// TIA Portal V20 export
TYPE "type_emRelations_em5_sequence"
// stored: Access Published, Namespace Unit1
   STRUCT
      transferPnPLeft : Struct
         jobs : "LAF_typeJobs";
         sequence : "LAF_typeSequence";
         selectJobStatus { S7_SetPoint := 'True'} : Array[0..10] of "LAF_typeJobStatus";
         "step" : "LER_typeStep";
         jobInterface : Struct
            sideTapePICKJob2_A : "LER_typeJobInterface";
            hotPressLeftPLACEJob3_A : "LER_typeJobInterface";
            hotPressLeftPICKJob4_A : "LER_typeJobInterface";
            sideTapePICKJob5_B : "LER_typeJobInterface";
            hotPressRightPLACEJob6_B : "LER_typeJobInterface";
            hotPressRightPICKJob7_B : "LER_typeJobInterface";
            hipotThicknessPLACEJob9 : "LER_typeJobInterface";
         END_STRUCT;
         homeCheck : Struct
            waitPosPartNoDetect { ExternalWritable := 'False'} : Bool;
            waitPosPartDetect { ExternalWritable := 'False'} : Bool;
            sideTapePosPartNoDetect { ExternalWritable := 'False'} : Bool;
            sideTapePosPartDetect { ExternalWritable := 'False'} : Bool;
            hotPressLeftPosPartNoDetect { ExternalWritable := 'False'} : Bool;
            hotPressLeftPosPartDetect { ExternalWritable := 'False'} : Bool;
            hotPressRightPosPartNoDetect { ExternalWritable := 'False'} : Bool;
            hotPressRightPosPartDetect { ExternalWritable := 'False'} : Bool;
            hipotThicknessPosPartNoDetect { ExternalWritable := 'False'} : Bool;
            hipotThicknessPosPartDetect { ExternalWritable := 'False'} : Bool;
            defaultPosPartDetect : Bool;
            defaultPosPartNoDetect : Bool;
         END_STRUCT;
      END_STRUCT;
      transferPnPRight : Struct
         jobs : "LAF_typeJobs";
         sequence : "LAF_typeSequence";
         selectJobStatus { S7_SetPoint := 'True'} : Array[0..10] of "LAF_typeJobStatus";
         "step" : "LER_typeStep";
         jobInterface : Struct
            hipotThicknessPICKJob2 : "LER_typeJobInterface";
            visionPLACEJob3 : "LER_typeJobInterface";
            visionPICKJob4 : "LER_typeJobInterface";
            laserMarkPLACEJob5 : "LER_typeJobInterface";
            laserMarkPICKJob6 : "LER_typeJobInterface";
            weightCheckPLACEJob9 : "LER_typeJobInterface";
         END_STRUCT;
         homeCheck : Struct
            waitPosPartNoDetect { ExternalWritable := 'False'} : Bool;
            waitPosPartDetect { ExternalWritable := 'False'} : Bool;
            hipotThicknessPosPartNoDetect { ExternalWritable := 'False'} : Bool;
            hipotThicknessPosPartDetect { ExternalWritable := 'False'} : Bool;
            visionPosPartNoDetect { ExternalWritable := 'False'} : Bool;
            visionPosPartDetect { ExternalWritable := 'False'} : Bool;
            laserMarkPosPartNoDetect { ExternalWritable := 'False'} : Bool;
            laserMarkPosPartDetect { ExternalWritable := 'False'} : Bool;
            weightCheckPosPartNoDetect { ExternalWritable := 'False'} : Bool;
            weightCheckPosPartDetect { ExternalWritable := 'False'} : Bool;
            defaultPosPartDetect : Bool;
            defaultPosPartNoDetect : Bool;
         END_STRUCT;
      END_STRUCT;
      GRnR_TransferPnP : Struct
         jobs : "LAF_typeJobs";
         sequence : "LAF_typeSequence";
         selectJobStatus { S7_SetPoint := 'True'} : Array[0..10] of "LAF_typeJobStatus";
         "step" : "LER_typeStep";
         jobInterface : Struct
            transferPnPLeft : Struct
               sideTapePICKJob2 : "LER_typeJobInterface";
               hipotThicknessPLACEJob3 : "LER_typeJobInterface";
               hipotThicknessPICKJob4 : "LER_typeJobInterface";
            END_STRUCT;
            transferPnPRight : Struct
               hipotThicknessPICKJob5 : "LER_typeJobInterface";
               visionPLACEJob6 : "LER_typeJobInterface";
               visionPICKJob7 : "LER_typeJobInterface";
               weightCheckPLACEJob8 : "LER_typeJobInterface";
               weightCheckPICKJob9 : "LER_typeJobInterface";
            END_STRUCT;
         END_STRUCT;
      END_STRUCT;
   END_STRUCT;
   // // transferPnPLeft."step".action1[101] : Step[101] : JOB[1] Condition
   // // transferPnPLeft."step".action1[110] : Step[110] : Transfer PP Left Clamp Open
   // // transferPnPLeft."step".action1[130] : Step[130] : Transfer PP Left Clamp Close
   // // transferPnPLeft."step".action1[160] : Step[160] : Transfer PP Left Y-Axis Wait Pos
   // // transferPnPLeft."step".action1[170] : Step[170] : Transfer PP Left Z-Axis Wait Pos
   // // transferPnPLeft."step".action1[180] : Step[180] : Transfer PP Left X-Axis Wait Pos
   // // transferPnPLeft."step".action1[190] : Step[190] : JOB[1] Step End
   // // transferPnPLeft."step".action1[201] : Step[201] : JOB[2] Condition
   // // transferPnPLeft."step".action1[210] : Step[210] : Transfer PP Left X/Z-Axis Side Tape Pos
   // // transferPnPLeft."step".action1[230] : Step[230] : Transfer PP Left Y-Axis Side Tape Pos
   // // transferPnPLeft."step".action1[240] : Step[240] : Transfer PP Left Clamp Close
   // // transferPnPLeft."step".action1[242] : Step[242] : Transfer PP Left [Unclamp request] => Side Tape Fix Stage
   // // transferPnPLeft."step".action1[280] : Step[280] : Transfer PP Left Y-Axis Wait Pos
   // // transferPnPLeft."step".action1[290] : Step[290] : JOB[2] Step End
   // // transferPnPLeft."step".action1[301] : Step[301] : JOB[3] Condition
   // // transferPnPLeft."step".action1[310] : Step[310] : Transfer PP Left X/Z-Axis Hot Press Left Pos
   // // transferPnPLeft."step".action1[330] : Step[330] : Transfer PP Left Y-Axis Hot Press Left Pos
   // // transferPnPLeft."step".action1[340] : Step[340] : Transfer PP Left [Lift Up Request] => Hot Press Left
   // // transferPnPLeft."step".action1[350] : Step[350] : Transfer PP Left Clamp Open
   // // transferPnPLeft."step".action1[380] : Step[380] : Transfer PP Left Y-Axis Wait Pos
   // // transferPnPLeft."step".action1[390] : Step[390] : JOB[3] Step End
   // // transferPnPLeft."step".action1[401] : Step[401] : JOB[4] Condition
   // // transferPnPLeft."step".action1[410] : Step[410] : Transfer PP Left X/Z-Axis Hot Press Left Pos
   // // transferPnPLeft."step".action1[430] : Step[430] : Transfer PP Left Y-Axis Hot Press Left Pos
   // // transferPnPLeft."step".action1[440] : Step[440] : Transfer PP Left Clamp Close
   // // transferPnPLeft."step".action1[480] : Step[480] : Transfer PP Left Y-Axis Wait Pos
   // // transferPnPLeft."step".action1[490] : Step[490] : JOB[4] Step End
   // // transferPnPLeft."step".action1[501] : Step[501] : JOB[5] Condition
   // // transferPnPLeft."step".action1[510] : Step[510] : Transfer PP Left X/Z-Axis Side Tape Pos
   // // transferPnPLeft."step".action1[530] : Step[530] : Transfer PP Left Y-Axis Side Tape Pos
   // // transferPnPLeft."step".action1[540] : Step[540] : Transfer PP Left Clamp Close
   // // transferPnPLeft."step".action1[542] : Step[542] : Transfer PP Left [Unclamp request] => Side Tape Fix Stage
   // // transferPnPLeft."step".action1[580] : Step[580] : Transfer PP Left Y-Axis Wait Pos
   // // transferPnPLeft."step".action1[590] : Step[590] : JOB[5] Step End
   // // transferPnPLeft."step".action1[601] : Step[601] : JOB[6] Condition
   // // transferPnPLeft."step".action1[610] : Step[610] : Transfer PP Left X/Z-Axis Hot Press Right Pos
   // // transferPnPLeft."step".action1[630] : Step[630] : Transfer PP Left Y-Axis Hot Press Right Pos
   // // transferPnPLeft."step".action1[640] : Step[640] : Transfer PP Left [Lift Up Request] => Hot Press Right
   // // transferPnPLeft."step".action1[650] : Step[650] : Transfer PP Left Clamp Open
   // // transferPnPLeft."step".action1[680] : Step[680] : Transfer PP Left Y-Axis Wait Pos
   // // transferPnPLeft."step".action1[690] : Step[690] : JOB[6] Step End
   // // transferPnPLeft."step".action1[701] : Step[701] : JOB[7] Condition
   // // transferPnPLeft."step".action1[710] : Step[710] : Transfer PP Left X/Z-Axis Hot Press Right Pos
   // // transferPnPLeft."step".action1[730] : Step[730] : Transfer PP Left Y-Axis Hot Press Right Pos
   // // transferPnPLeft."step".action1[740] : Step[740] : Transfer PP Left Clamp Close
   // // transferPnPLeft."step".action1[780] : Step[780] : Transfer PP Left Y-Axis Wait Pos
   // // transferPnPLeft."step".action1[790] : Step[790] : JOB[7] Step End
   // // transferPnPLeft."step".action1[901] : Step[901] : JOB[9] Condition
   // // transferPnPLeft."step".action1[910] : Step[910] : Transfer PP Left X/Z-Axis Hipot & Thickness Pos
   // // transferPnPLeft."step".action1[930] : Step[930] : Transfer PP Left Y-Axis Hipot & Thickness Pos
   // // transferPnPLeft."step".action1[940] : Step[940] : Transfer PP Left [Lift Up Request] => Hipot & Thickness
   // // transferPnPLeft."step".action1[950] : Step[950] : Transfer PP Left Clamp Open
   // // transferPnPLeft."step".action1[980] : Step[980] : Transfer PP Left Y-Axis Wait Pos
   // // transferPnPLeft."step".action1[981] : Step[981] : Transfer PP Left X/Z-Axis Wait Pos
   // // transferPnPLeft."step".action1[990] : Step[990] : JOB[9] Step End
   // // transferPnPLeft."step".transition1[101] : Step[101] : JOB[1] Condition
   // // transferPnPLeft."step".transition1[110] : Step[110] : Transfer PP Left Clamp Open
   // // transferPnPLeft."step".transition1[130] : Step[130] : Transfer PP Left Clamp Close
   // // transferPnPLeft."step".transition1[160] : Step[160] : Transfer PP Left Y-Axis Wait Pos
   // // transferPnPLeft."step".transition1[170] : Step[170] : Transfer PP Left Z-Axis Wait Pos
   // // transferPnPLeft."step".transition1[180] : Step[180] : Transfer PP Left X-Axis Wait Pos
   // // transferPnPLeft."step".transition1[190] : Step[190] : JOB[1] Step End
   // // transferPnPLeft."step".transition1[201] : Step[201] : JOB[2] Condition
   // // transferPnPLeft."step".transition1[210] : Step[210] : Transfer PP Left X/Z-Axis Side Tape Pos
   // // transferPnPLeft."step".transition1[230] : Step[230] : Transfer PP Left Y-Axis Side Tape Pos
   // // transferPnPLeft."step".transition1[240] : Step[240] : Transfer PP Left Clamp Close
   // // transferPnPLeft."step".transition1[242] : Step[242] : Transfer PP Left [Unclamp request] => Side Tape Fix Stage
   // // transferPnPLeft."step".transition1[280] : Step[280] : Transfer PP Left Y-Axis Wait Pos
   // // transferPnPLeft."step".transition1[290] : Step[290] : JOB[2] Step End
   // // transferPnPLeft."step".transition1[301] : Step[301] : JOB[3] Condition
   // // transferPnPLeft."step".transition1[310] : Step[310] : Transfer PP Left X/Z-Axis Hot Press Left Pos
   // // transferPnPLeft."step".transition1[330] : Step[330] : Transfer PP Left Y-Axis Hot Press Left Pos
   // // transferPnPLeft."step".transition1[340] : Step[340] : Transfer PP Left [Lift Up Request] => Hot Press Left
   // // transferPnPLeft."step".transition1[350] : Step[350] : Transfer PP Left Clamp Open
   // // transferPnPLeft."step".transition1[380] : Step[380] : Transfer PP Left Y-Axis Wait Pos
   // // transferPnPLeft."step".transition1[390] : Step[390] : JOB[3] Step End
   // // transferPnPLeft."step".transition1[401] : Step[401] : JOB[4] Condition
   // // transferPnPLeft."step".transition1[410] : Step[410] : Transfer PP Left X/Z-Axis Hot Press Left Pos
   // // transferPnPLeft."step".transition1[430] : Step[430] : Transfer PP Left Y-Axis Hot Press Left Pos
   // // transferPnPLeft."step".transition1[440] : Step[440] : Transfer PP Left Clamp Close
   // // transferPnPLeft."step".transition1[480] : Step[480] : Transfer PP Left Y-Axis Wait Pos
   // // transferPnPLeft."step".transition1[490] : Step[490] : JOB[4] Step End
   // // transferPnPLeft."step".transition1[501] : Step[501] : JOB[5] Condition
   // // transferPnPLeft."step".transition1[510] : Step[510] : Transfer PP Left X/Z-Axis Side Tape Pos
   // // transferPnPLeft."step".transition1[530] : Step[530] : Transfer PP Left Y-Axis Side Tape Pos
   // // transferPnPLeft."step".transition1[540] : Step[540] : Transfer PP Left Clamp Close
   // // transferPnPLeft."step".transition1[542] : Step[542] : Transfer PP Left [Unclamp request] => Side Tape Fix Stage
   // // transferPnPLeft."step".transition1[580] : Step[580] : Transfer PP Left Y-Axis Wait Pos
   // // transferPnPLeft."step".transition1[590] : Step[590] : JOB[5] Step End
   // // transferPnPLeft."step".transition1[601] : Step[601] : JOB[6] Condition
   // // transferPnPLeft."step".transition1[610] : Step[610] : Transfer PP Left X/Z-Axis Hot Press Right Pos
   // // transferPnPLeft."step".transition1[630] : Step[630] : Transfer PP Left Y-Axis Hot Press Right Pos
   // // transferPnPLeft."step".transition1[640] : Step[640] : Transfer PP Left [Lift Up Request] => Hot Press Right
   // // transferPnPLeft."step".transition1[650] : Step[650] : Transfer PP Left Clamp Open
   // // transferPnPLeft."step".transition1[680] : Step[680] : Transfer PP Left Y-Axis Wait Pos
   // // transferPnPLeft."step".transition1[690] : Step[690] : JOB[6] Step End
   // // transferPnPLeft."step".transition1[701] : Step[701] : JOB[7] Condition
   // // transferPnPLeft."step".transition1[710] : Step[710] : Transfer PP Left X/Z-Axis Hot Press Right Pos
   // // transferPnPLeft."step".transition1[730] : Step[730] : Transfer PP Left Y-Axis Hot Press Right Pos
   // // transferPnPLeft."step".transition1[740] : Step[740] : Transfer PP Left Clamp Close
   // // transferPnPLeft."step".transition1[780] : Step[780] : Transfer PP Left Y-Axis Wait Pos
   // // transferPnPLeft."step".transition1[790] : Step[790] : JOB[7] Step End
   // // transferPnPLeft."step".transition1[901] : Step[901] : JOB[9] Condition
   // // transferPnPLeft."step".transition1[910] : Step[910] : Transfer PP Left X/Z-Axis Hipot & Thickness Pos
   // // transferPnPLeft."step".transition1[930] : Step[930] : Transfer PP Left Y-Axis Hipot & Thickness Pos
   // // transferPnPLeft."step".transition1[940] : Step[940] : Transfer PP Left [Lift Up Request] => Hipot & Thickness
   // // transferPnPLeft."step".transition1[950] : Step[950] : Transfer PP Left Clamp Open
   // // transferPnPLeft."step".transition1[980] : Step[980] : Transfer PP Left Y-Axis Wait Pos
   // // transferPnPLeft."step".transition1[981] : Step[981] : Transfer PP Left X/Z-Axis Wait Pos
   // // transferPnPLeft."step".transition1[990] : Step[990] : JOB[9] Step End
   // // transferPnPRight."step".action1[101] : Step[101] : JOB[1] Condition
   // // transferPnPRight."step".action1[110] : Step[110] : Transfer PP Right Clamp Open
   // // transferPnPRight."step".action1[130] : Step[130] : Transfer PP Right Clamp Close
   // // transferPnPRight."step".action1[160] : Step[160] : Transfer PP Right Y-Axis Wait Position
   // // transferPnPRight."step".action1[170] : Step[170] : Transfer PP Right Z-Axis Wait Position
   // // transferPnPRight."step".action1[180] : Step[180] : Transfer PP Right X-Axis Wait Position
   // // transferPnPRight."step".action1[190] : Step[190] : JOB[1] Step End
   // // transferPnPRight."step".action1[201] : Step[201] : JOB[2] Condition
   // // transferPnPRight."step".action1[210] : Step[210] : Transfer PP Right X/Z-Axis Hipot & Thickness Pos
   // // transferPnPRight."step".action1[230] : Step[230] : Transfer PP Right Y-Axis Hipot & Thickness Pos
   // // transferPnPRight."step".action1[240] : Step[240] : Transfer PP Right Clamp Close
   // // transferPnPRight."step".action1[280] : Step[280] : Transfer PP Right Y-Axis Wait Pos
   // // transferPnPRight."step".action1[290] : Step[290] : JOB[2] Step End
   // // transferPnPRight."step".action1[301] : Step[301] : JOB[3] Condition
   // // transferPnPRight."step".action1[310] : Step[310] : Transfer PP Right X/Z-Axis Vision Pos
   // // transferPnPRight."step".action1[330] : Step[330] : Transfer PP Right Y-Axis Vision Pos
   // // transferPnPRight."step".action1[340] : Step[340] : Transfer PP Right [Lift Up Request] => Vision Check
   // // transferPnPRight."step".action1[350] : Step[350] : Transfer PP Right Clamp Open
   // // transferPnPRight."step".action1[380] : Step[380] : Transfer PP Right Y-Axis Wait Pos
   // // transferPnPRight."step".action1[390] : Step[390] : JOB[3] Step End
   // // transferPnPRight."step".action1[401] : Step[401] : JOB[4] Condition
   // // transferPnPRight."step".action1[410] : Step[410] : Transfer PP Right X/Z-Axis Vision Pos
   // // transferPnPRight."step".action1[430] : Step[430] : Transfer PP Right Y-Axis Vision Pos
   // // transferPnPRight."step".action1[440] : Step[440] : Transfer PP Right Clamp Close
   // // transferPnPRight."step".action1[480] : Step[480] : Transfer PP Right Y-Axis Wait Pos
   // // transferPnPRight."step".action1[490] : Step[490] : JOB[4] Step End
   // // transferPnPRight."step".action1[501] : Step[501] : JOB[5] Condition
   // // transferPnPRight."step".action1[510] : Step[510] : Transfer PP Right X/Z-Axis Laser Mark Pos
   // // transferPnPRight."step".action1[530] : Step[530] : Transfer PP Right Y-Axis Laser Mark Pos
   // // transferPnPRight."step".action1[540] : Step[540] : Transfer PP Right [Lift Up Request] => Laser Mark
   // // transferPnPRight."step".action1[550] : Step[550] : Transfer PP Right Clamp Open
   // // transferPnPRight."step".action1[580] : Step[580] : Transfer PP Right Y-Axis Wait Pos
   // // transferPnPRight."step".action1[590] : Step[590] : JOB[5] Step End
   // // transferPnPRight."step".action1[601] : Step[601] : JOB[6] Condition
   // // transferPnPRight."step".action1[602] : Step[602] : QR Read Start
   // // transferPnPRight."step".action1[603] : Step[603] : QR Read Result
   // // transferPnPRight."step".action1[604] : Step[604] : QR Read Start [NG]
   // // transferPnPRight."step".action1[605] : Step[605] : QR Read Result [NG]
   // // transferPnPRight."step".action1[610] : Step[610] : Transfer PP Right X/Z-Axis Laser Mark Pos
   // // transferPnPRight."step".action1[630] : Step[630] : Transfer PP Right Y-Axis Laser Mark Pos
   // // transferPnPRight."step".action1[640] : Step[640] : Transfer PP Right Clamp Close
   // // transferPnPRight."step".action1[680] : Step[680] : Transfer PP Right Y-Axis Wait Pos
   // // transferPnPRight."step".action1[690] : Step[690] : JOB[6] Step End
   // // transferPnPRight."step".action1[701] : Step[701] : JOB[7] Condition
   // // transferPnPRight."step".action1[710] : Step[710] : Transfer PP Right X/Z-Axis Laser Mark Pos
   // // transferPnPRight."step".action1[730] : Step[730] : Transfer PP Right Y-Axis Laser Mark Pos
   // // transferPnPRight."step".action1[740] : Step[740] : Transfer PP Right [Lift Up Request] => Laser Mark
   // // transferPnPRight."step".action1[750] : Step[750] : Transfer PP Right Clamp Open
   // // transferPnPRight."step".action1[780] : Step[780] : Transfer PP Right Y-Axis Wait Pos
   // // transferPnPRight."step".action1[790] : Step[790] : JOB[7] Step End
   // // transferPnPRight."step".action1[801] : Step[801] : JOB[8] Condition
   // // transferPnPRight."step".action1[810] : Step[810] : Transfer PP Right X/Z-Axis Laser Mark Pos
   // // transferPnPRight."step".action1[830] : Step[830] : Transfer PP Right Y-Axis Laser Mark Pos
   // // transferPnPRight."step".action1[840] : Step[840] : Transfer PP Right Clamp Close
   // // transferPnPRight."step".action1[880] : Step[880] : Transfer PP Right Y-Axis Wait Pos
   // // transferPnPRight."step".action1[890] : Step[890] : JOB[8] Step End
   // // transferPnPRight."step".action1[901] : Step[901] : JOB[9] Condition
   // // transferPnPRight."step".action1[910] : Step[910] : Transfer PP Right X/Z-Axis Weight Check Pos
   // // transferPnPRight."step".action1[930] : Step[930] : Transfer PP Right Y-Axis Weight Check Pos
   // // transferPnPRight."step".action1[931] : Step[931] : Transfer PP Right Z-Axis Weight Check Pos
   // // transferPnPRight."step".action1[940] : Step[940] : Transfer PP Right [Lift Up Request] => Weight Check
   // // transferPnPRight."step".action1[950] : Step[950] : Transfer PP Right Clamp Open
   // // transferPnPRight."step".action1[980] : Step[980] : Transfer PP Right Y-Axis Wait Pos
   // // transferPnPRight."step".action1[981] : Step[981] : Transfer PP Right X/Z-Axis Wait Pos
   // // transferPnPRight."step".action1[990] : Step[990] : JOB[9] Step End
   // // transferPnPRight."step".transition1[101] : Step[101] : JOB[1] Condition
   // // transferPnPRight."step".transition1[110] : Step[110] : Transfer PP Right Clamp Open
   // // transferPnPRight."step".transition1[130] : Step[130] : Transfer PP Right Clamp Close
   // // transferPnPRight."step".transition1[160] : Step[160] : Transfer PP Right Y-Axis Wait Position
   // // transferPnPRight."step".transition1[170] : Step[170] : Transfer PP Right Z-Axis Wait Position
   // // transferPnPRight."step".transition1[180] : Step[180] : Transfer PP Right X-Axis Wait Position
   // // transferPnPRight."step".transition1[190] : Step[190] : JOB[1] Step End
   // // transferPnPRight."step".transition1[201] : Step[201] : JOB[2] Condition
   // // transferPnPRight."step".transition1[210] : Step[210] : Transfer PP Right X/Z-Axis Hipot & Thickness Pos
   // // transferPnPRight."step".transition1[230] : Step[230] : Transfer PP Right Y-Axis Hipot & Thickness Pos
   // // transferPnPRight."step".transition1[240] : Step[240] : Transfer PP Right Clamp Close
   // // transferPnPRight."step".transition1[280] : Step[280] : Transfer PP Right Y-Axis Wait Pos
   // // transferPnPRight."step".transition1[290] : Step[290] : JOB[2] Step End
   // // transferPnPRight."step".transition1[301] : Step[301] : JOB[3] Condition
   // // transferPnPRight."step".transition1[310] : Step[310] : Transfer PP Right X/Z-Axis Vision Pos
   // // transferPnPRight."step".transition1[330] : Step[330] : Transfer PP Right Y-Axis Vision Pos
   // // transferPnPRight."step".transition1[340] : Step[340] : Transfer PP Right [Lift Up Request] => Vision Check
   // // transferPnPRight."step".transition1[350] : Step[350] : Transfer PP Right Clamp Open
   // // transferPnPRight."step".transition1[380] : Step[380] : Transfer PP Right Y-Axis Wait Pos
   // // transferPnPRight."step".transition1[390] : Step[390] : JOB[3] Step End
   // // transferPnPRight."step".transition1[401] : Step[401] : JOB[4] Condition
   // // transferPnPRight."step".transition1[410] : Step[410] : Transfer PP Right X/Z-Axis Vision Pos
   // // transferPnPRight."step".transition1[430] : Step[430] : Transfer PP Right Y-Axis Vision Pos
   // // transferPnPRight."step".transition1[440] : Step[440] : Transfer PP Right Clamp Close
   // // transferPnPRight."step".transition1[480] : Step[480] : Transfer PP Right Y-Axis Wait Pos
   // // transferPnPRight."step".transition1[490] : Step[490] : JOB[4] Step End
   // // transferPnPRight."step".transition1[501] : Step[501] : JOB[5] Condition
   // // transferPnPRight."step".transition1[510] : Step[510] : Transfer PP Right X/Z-Axis Laser Mark Pos
   // // transferPnPRight."step".transition1[530] : Step[530] : Transfer PP Right Y-Axis Laser Mark Pos
   // // transferPnPRight."step".transition1[540] : Step[540] : Transfer PP Right [Lift Up Request] => Laser Mark
   // // transferPnPRight."step".transition1[550] : Step[550] : Transfer PP Right Clamp Open
   // // transferPnPRight."step".transition1[580] : Step[580] : Transfer PP Right Y-Axis Wait Pos
   // // transferPnPRight."step".transition1[590] : Step[590] : JOB[5] Step End
   // // transferPnPRight."step".transition1[601] : Step[601] : JOB[6] Condition
   // // transferPnPRight."step".transition1[602] : Step[602] : QR Read Start
   // // transferPnPRight."step".transition1[603] : Step[603] : QR Read Result
   // // transferPnPRight."step".transition1[604] : Step[604] : QR Read Start [NG]
   // // transferPnPRight."step".transition1[605] : Step[605] : QR Read Result [NG]
   // // transferPnPRight."step".transition1[610] : Step[610] : Transfer PP Right X/Z-Axis Laser Mark Pos
   // // transferPnPRight."step".transition1[630] : Step[630] : Transfer PP Right Y-Axis Laser Mark Pos
   // // transferPnPRight."step".transition1[640] : Step[640] : Transfer PP Right Clamp Close
   // // transferPnPRight."step".transition1[680] : Step[680] : Transfer PP Right Y-Axis Wait Pos
   // // transferPnPRight."step".transition1[690] : Step[690] : JOB[6] Step End
   // // transferPnPRight."step".transition1[701] : Step[701] : JOB[7] Condition
   // // transferPnPRight."step".transition1[710] : Step[710] : Transfer PP Right X/Z-Axis Laser Mark Pos
   // // transferPnPRight."step".transition1[730] : Step[730] : Transfer PP Right Y-Axis Laser Mark Pos
   // // transferPnPRight."step".transition1[740] : Step[740] : Transfer PP Right [Lift Up Request] => Laser Mark
   // // transferPnPRight."step".transition1[750] : Step[750] : Transfer PP Right Clamp Open
   // // transferPnPRight."step".transition1[780] : Step[780] : Transfer PP Right Y-Axis Wait Pos
   // // transferPnPRight."step".transition1[790] : Step[790] : JOB[7] Step End
   // // transferPnPRight."step".transition1[801] : Step[801] : JOB[8] Condition
   // // transferPnPRight."step".transition1[810] : Step[810] : Transfer PP Right X/Z-Axis Laser Mark Pos
   // // transferPnPRight."step".transition1[830] : Step[830] : Transfer PP Right Y-Axis Laser Mark Pos
   // // transferPnPRight."step".transition1[840] : Step[840] : Transfer PP Right Clamp Close
   // // transferPnPRight."step".transition1[880] : Step[880] : Transfer PP Right Y-Axis Wait Pos
   // // transferPnPRight."step".transition1[890] : Step[890] : JOB[8] Step End
   // // transferPnPRight."step".transition1[901] : Step[901] : JOB[9] Condition
   // // transferPnPRight."step".transition1[910] : Step[910] : Transfer PP Right X/Z-Axis Weight Check Pos
   // // transferPnPRight."step".transition1[930] : Step[930] : Transfer PP Right Y-Axis Weight Check Pos
   // // transferPnPRight."step".transition1[931] : Step[931] : Transfer PP Right Z-Axis Weight Check Pos
   // // transferPnPRight."step".transition1[940] : Step[940] : Transfer PP Right [Lift Up Request] => Weight Check
   // // transferPnPRight."step".transition1[950] : Step[950] : Transfer PP Right Clamp Open
   // // transferPnPRight."step".transition1[980] : Step[980] : Transfer PP Right Y-Axis Wait Pos
   // // transferPnPRight."step".transition1[981] : Step[981] : Transfer PP Right X/Z-Axis Wait Pos
   // // transferPnPRight."step".transition1[990] : Step[990] : JOB[9] Step End
   // // GRnR_TransferPnP."step".action1[201] : Step[201] : JOB[2] Condition
   // // GRnR_TransferPnP."step".action1[210] : Step[210] : Transfer PP Left X/Z-Axis Side Tape Pos
   // // GRnR_TransferPnP."step".action1[230] : Step[230] : Transfer PP Left Y-Axis Side Tape Pos
   // // GRnR_TransferPnP."step".action1[240] : Step[240] : Transfer PP Left Clamp Close
   // // GRnR_TransferPnP."step".action1[241] : Step[241] : Transfer PP Left [Unclamp request] => Side Tape Fix Stage
   // // GRnR_TransferPnP."step".action1[280] : Step[280] : Transfer PP Left Y-Axis Wait Pos
   // // GRnR_TransferPnP."step".action1[290] : Step[290] : JOB[2] Step End
   // // GRnR_TransferPnP."step".action1[301] : Step[301] : JOB[3] Condition
   // // GRnR_TransferPnP."step".action1[310] : Step[310] : Transfer PP Left X/Z-Axis Hipot & Thickness Pos
   // // GRnR_TransferPnP."step".action1[330] : Step[330] : Transfer PP Left Y-Axis Hipot & Thickness Pos
   // // GRnR_TransferPnP."step".action1[340] : Step[340] : Transfer PP Left [Lift Up Request] => Hipot & Thickness
   // // GRnR_TransferPnP."step".action1[350] : Step[350] : Transfer PP Left Clamp Open
   // // GRnR_TransferPnP."step".action1[380] : Step[380] : Transfer PP Left Y-Axis Wait Pos
   // // GRnR_TransferPnP."step".action1[381] : Step[381] : Transfer PP Left X/Z-Axis Wait Pos
   // // GRnR_TransferPnP."step".action1[390] : Step[390] : JOB[3] Step End
   // // GRnR_TransferPnP."step".action1[401] : Step[401] : JOB[4] Condition
   // // GRnR_TransferPnP."step".action1[410] : Step[410] : Transfer PP Left X/Z-Axis Hipot & Thickness Pos
   // // GRnR_TransferPnP."step".action1[430] : Step[430] : Transfer PP Left Y-Axis Hipot & Thickness Pos
   // // GRnR_TransferPnP."step".action1[440] : Step[440] : Transfer PP Left Clamp Close
   // // GRnR_TransferPnP."step".action1[480] : Step[480] : Transfer PP Left Y-Axis Wait Pos
   // // GRnR_TransferPnP."step".action1[481] : Step[481] : Transfer PP Left X/Z-Axis Wait Pos
   // // GRnR_TransferPnP."step".action1[490] : Step[490] : JOB[4] Step End
   // // GRnR_TransferPnP."step".action1[501] : Step[501] : JOB[5] Condition
   // // GRnR_TransferPnP."step".action1[510] : Step[510] : Transfer PP Right X/Z-Axis Hipot & Thickness Pos
   // // GRnR_TransferPnP."step".action1[530] : Step[530] : Transfer PP Right Y-Axis Hipot & Thickness Pos
   // // GRnR_TransferPnP."step".action1[540] : Step[540] : Transfer PP Right Clamp Close
   // // GRnR_TransferPnP."step".action1[580] : Step[580] : Transfer PP Right Y-Axis Wait Pos
   // // GRnR_TransferPnP."step".action1[590] : Step[590] : JOB[5] Step End
   // // GRnR_TransferPnP."step".action1[601] : Step[601] : JOB[6] Condition
   // // GRnR_TransferPnP."step".action1[610] : Step[610] : Transfer PP Right X/Z-Axis Vision Pos
   // // GRnR_TransferPnP."step".action1[630] : Step[630] : Transfer PP Right Y-Axis Vision Pos
   // // GRnR_TransferPnP."step".action1[640] : Step[640] : Transfer PP Right [Lift Up Request] => Vision Check
   // // GRnR_TransferPnP."step".action1[650] : Step[650] : Transfer PP Right Clamp Open
   // // GRnR_TransferPnP."step".action1[680] : Step[680] : Transfer PP Right Y-Axis Wait Pos
   // // GRnR_TransferPnP."step".action1[690] : Step[690] : JOB[6] Step End
   // // GRnR_TransferPnP."step".action1[701] : Step[701] : JOB[7] Condition
   // // GRnR_TransferPnP."step".action1[710] : Step[710] : Transfer PP Right X/Z-Axis Vision Pos
   // // GRnR_TransferPnP."step".action1[730] : Step[730] : Transfer PP Right Y-Axis Vision Pos
   // // GRnR_TransferPnP."step".action1[740] : Step[740] : Transfer PP Right Clamp Close
   // // GRnR_TransferPnP."step".action1[780] : Step[780] : Transfer PP Right Y-Axis Wait Pos
   // // GRnR_TransferPnP."step".action1[790] : Step[790] : JOB[7] Step End
   // // GRnR_TransferPnP."step".action1[801] : Step[801] : JOB[8] Condition
   // // GRnR_TransferPnP."step".action1[810] : Step[810] : Transfer PP Right X/Z-Axis Weight Check Pos
   // // GRnR_TransferPnP."step".action1[830] : Step[830] : Transfer PP Right Y-Axis Weight Check Pos
   // // GRnR_TransferPnP."step".action1[831] : Step[831] : Transfer PP Right Z-Axis Weight Check Pos
   // // GRnR_TransferPnP."step".action1[840] : Step[840] : Transfer PP Right [Lift Up Request] => Weight Check
   // // GRnR_TransferPnP."step".action1[850] : Step[850] : Transfer PP Right Clamp Open
   // // GRnR_TransferPnP."step".action1[880] : Step[880] : Transfer PP Right Y-Axis Wait Pos
   // // GRnR_TransferPnP."step".action1[881] : Step[881] : Transfer PP Right X/Z-Axis Wait Pos
   // // GRnR_TransferPnP."step".action1[890] : Step[890] : JOB[8] Step End
   // // GRnR_TransferPnP."step".action1[901] : Step[901] : JOB[9] Condition
   // // GRnR_TransferPnP."step".action1[910] : Step[910] : Transfer PP Right X/Z-Axis Weight Check Pos
   // // GRnR_TransferPnP."step".action1[930] : Step[930] : Transfer PP Right Y-Axis Weight Pos
   // // GRnR_TransferPnP."step".action1[940] : Step[940] : Transfer PP Right Clamp Close
   // // GRnR_TransferPnP."step".transition1[201] : Step[201] : JOB[2] Condition
   // // GRnR_TransferPnP."step".transition1[210] : Step[210] : Transfer PP Left X/Z-Axis Side Tape Pos
   // // GRnR_TransferPnP."step".transition1[230] : Step[230] : Transfer PP Left Y-Axis Side Tape Pos
   // // GRnR_TransferPnP."step".transition1[240] : Step[240] : Transfer PP Left Clamp Close
   // // GRnR_TransferPnP."step".transition1[241] : Step[241] : Transfer PP Left [Unclamp request] => Side Tape Fix Stage
   // // GRnR_TransferPnP."step".transition1[280] : Step[280] : Transfer PP Left Y-Axis Wait Pos
   // // GRnR_TransferPnP."step".transition1[290] : Step[290] : JOB[2] Step End
   // // GRnR_TransferPnP."step".transition1[301] : Step[301] : JOB[3] Condition
   // // GRnR_TransferPnP."step".transition1[310] : Step[310] : Transfer PP Left X/Z-Axis Hipot & Thickness Pos
   // // GRnR_TransferPnP."step".transition1[330] : Step[330] : Transfer PP Left Y-Axis Hipot & Thickness Pos
   // // GRnR_TransferPnP."step".transition1[340] : Step[340] : Transfer PP Left [Lift Up Request] => Hipot & Thickness
   // // GRnR_TransferPnP."step".transition1[350] : Step[350] : Transfer PP Left Clamp Open
   // // GRnR_TransferPnP."step".transition1[380] : Step[380] : Transfer PP Left Y-Axis Wait Pos
   // // GRnR_TransferPnP."step".transition1[381] : Step[381] : Transfer PP Left X/Z-Axis Wait Pos
   // // GRnR_TransferPnP."step".transition1[390] : Step[390] : JOB[3] Step End
   // // GRnR_TransferPnP."step".transition1[401] : Step[401] : JOB[4] Condition
   // // GRnR_TransferPnP."step".transition1[410] : Step[410] : Transfer PP Left X/Z-Axis Hipot & Thickness Pos
   // // GRnR_TransferPnP."step".transition1[430] : Step[430] : Transfer PP Left Y-Axis Hipot & Thickness Pos
   // // GRnR_TransferPnP."step".transition1[440] : Step[440] : Transfer PP Left Clamp Close
   // // GRnR_TransferPnP."step".transition1[480] : Step[480] : Transfer PP Left Y-Axis Wait Pos
   // // GRnR_TransferPnP."step".transition1[481] : Step[481] : Transfer PP Left X/Z-Axis Wait Pos
   // // GRnR_TransferPnP."step".transition1[490] : Step[490] : JOB[4] Step End
   // // GRnR_TransferPnP."step".transition1[501] : Step[501] : JOB[5] Condition
   // // GRnR_TransferPnP."step".transition1[510] : Step[510] : Transfer PP Right X/Z-Axis Hipot & Thickness Pos
   // // GRnR_TransferPnP."step".transition1[530] : Step[530] : Transfer PP Right Y-Axis Hipot & Thickness Pos
   // // GRnR_TransferPnP."step".transition1[540] : Step[540] : Transfer PP Right Clamp Close
   // // GRnR_TransferPnP."step".transition1[580] : Step[580] : Transfer PP Right Y-Axis Wait Pos
   // // GRnR_TransferPnP."step".transition1[590] : Step[590] : JOB[5] Step End
   // // GRnR_TransferPnP."step".transition1[601] : Step[601] : JOB[6] Condition
   // // GRnR_TransferPnP."step".transition1[610] : Step[610] : Transfer PP Right X/Z-Axis Vision Pos
   // // GRnR_TransferPnP."step".transition1[630] : Step[630] : Transfer PP Right Y-Axis Vision Pos
   // // GRnR_TransferPnP."step".transition1[640] : Step[640] : Transfer PP Right [Lift Up Request] => Vision Check
   // // GRnR_TransferPnP."step".transition1[650] : Step[650] : Transfer PP Right Clamp Open
   // // GRnR_TransferPnP."step".transition1[680] : Step[680] : Transfer PP Right Y-Axis Wait Pos
   // // GRnR_TransferPnP."step".transition1[690] : Step[690] : JOB[6] Step End
   // // GRnR_TransferPnP."step".transition1[701] : Step[701] : JOB[7] Condition
   // // GRnR_TransferPnP."step".transition1[710] : Step[710] : Transfer PP Right X/Z-Axis Vision Pos
   // // GRnR_TransferPnP."step".transition1[730] : Step[730] : Transfer PP Right Y-Axis Vision Pos
   // // GRnR_TransferPnP."step".transition1[740] : Step[740] : Transfer PP Right Clamp Close
   // // GRnR_TransferPnP."step".transition1[780] : Step[780] : Transfer PP Right Y-Axis Wait Pos
   // // GRnR_TransferPnP."step".transition1[790] : Step[790] : JOB[7] Step End
   // // GRnR_TransferPnP."step".transition1[801] : Step[801] : JOB[8] Condition
   // // GRnR_TransferPnP."step".transition1[810] : Step[810] : Transfer PP Right X/Z-Axis Weight Check Pos
   // // GRnR_TransferPnP."step".transition1[830] : Step[830] : Transfer PP Right Y-Axis Weight Check Pos
   // // GRnR_TransferPnP."step".transition1[831] : Step[831] : Transfer PP Right Z-Axis Weight Check Pos
   // // GRnR_TransferPnP."step".transition1[840] : Step[840] : Transfer PP Right [Lift Up Request] => Weight Check
   // // GRnR_TransferPnP."step".transition1[850] : Step[850] : Transfer PP Right Clamp Open
   // // GRnR_TransferPnP."step".transition1[880] : Step[880] : Transfer PP Right Y-Axis Wait Pos
   // // GRnR_TransferPnP."step".transition1[881] : Step[881] : Transfer PP Right X/Z-Axis Wait Pos
   // // GRnR_TransferPnP."step".transition1[890] : Step[890] : JOB[8] Step End
   // // GRnR_TransferPnP."step".transition1[901] : Step[901] : JOB[9] Condition
   // // GRnR_TransferPnP."step".transition1[910] : Step[910] : Transfer PP Right X/Z-Axis Weight Check Pos
   // // GRnR_TransferPnP."step".transition1[930] : Step[930] : Transfer PP Right Y-Axis Weight Pos
   // // GRnR_TransferPnP."step".transition1[940] : Step[940] : Transfer PP Right Clamp Close
END_TYPE
